Staubli VAL3: StaubliCalTool7.dtx

bool bFinish
bool bTeach1_1
bool bTeach1_2
bool bTeach1_3
bool bTeach1_4
bool bTeach2_2_1
bool bTeach2_2_2
bool bTeach2_3_1
bool bTeach2_3_2
bool bTeach2_3_3
bool bTeach3_1
bool bTeach3_2
public bool bUpLoad
configRx cConfigSame
jointRx jTest = {j1=43.06, j2=91.68, j3=-102.32, j4=-44.78, j5=56.91, j6=19.1}
mdesc mNomSpeed = {blend=cartesian}
mdesc mSlow = {vel=2, tmax=20, blend=cartesian, leave=0, reach=0}
mdesc mSpeed = {blend=cartesian, leave=0, reach=0}
num nMount = 1
num nOffsetRx
num nOffsetRy
num nOffsetRz
num nOffsetX
num nOffsetY
num nOffsetZ
num nS1[4]
num nS2[4]
num nS3[4]
num nS4[4]
num nScX
num nScY
num nScZ
pointRx p1_1 = {fatherId=world[0]}
pointRx p1_2 = {fatherId=world[0]}
pointRx p1_3 = {fatherId=world[0]}
pointRx p1_4 = {fatherId=world[0]}
pointRx p2_2_1 = {fatherId=world[0]}
pointRx p2_2_2 = {fatherId=world[0]}
pointRx p2_3_1 = {fatherId=world[0]}
pointRx p2_3_2 = {fatherId=world[0]}
pointRx p2_3_3 = {fatherId=world[0]}
pointRx p3_1 = {fatherId=world[0]}
pointRx p3_2 = {fatherId=world[0]}
pointRx pA = {x=1125.79, y=48.029029, z=-225.08575, rx=138.637496, ry=-37.318166, rz=51.328762, fatherId=world[0]}
pointRx pB = {x=1125.79, y=48.029029, z=-225.08575, rx=-41.362504, ry=-142.681834, rz=-38.671238, fatherId=world[0]}
pointRx pGoBack[11]
  [0] = {x=1244.112691, y=114.588869, z=210.083779, rx=0.001417, ry=-179.995766, rz=-83.364715, fatherId=world[0]}
  [1] = {x=1244.112692, y=114.588869, z=206.594488, rx=0.001253, ry=-179.995669, rz=-85.661401, fatherId=world[0]}
  [2] = {x=1244.112694, y=114.588869, z=203.105197, rx=0.001086, ry=-179.99558, rz=-87.958087, fatherId=world[0]}
  [3] = {x=1244.112696, y=114.588869, z=199.615906, rx=-179.999086, ry=-0.004503, rz=89.745227, fatherId=world[0]}
  [4] = {x=1244.112697, y=114.588869, z=196.126615, rx=-179.99926, ry=-0.004579, rz=87.448541, fatherId=world[0]}
  [5] = {x=1244.112699, y=114.588869, z=192.637324, rx=-179.999438, ry=-0.004648, rz=85.151855, fatherId=world[0]}
  [6] = {x=1244.1127, y=114.588869, z=189.148033, rx=-179.999618, ry=-0.00471, rz=82.855169, fatherId=world[0]}
  [7] = {x=1244.112702, y=114.588869, z=185.658742, rx=-179.9998, ry=-0.004765, rz=80.558483, fatherId=world[0]}
  [8] = {x=1244.112703, y=114.588869, z=182.169451, rx=-179.999984, ry=-0.004812, rz=78.261797, fatherId=world[0]}
  [9] = {x=1244.112705, y=114.588869, z=178.68016, rx=179.99983, ry=-0.004852, rz=75.965111, fatherId=world[0]}
  [10] = {x=1244.112706, y=114.588869, z=175.190869, rx=179.999642, ry=-0.004884, rz=73.668424, fatherId=world[0]}
pointRx pTraj = {x=1125.79, y=48.029029, z=-225.08575, rx=138.637496, ry=-37.318166, rz=42.328762, fatherId=world[0]}
string sLanguge = "Chinese"
string sMount = "floor"
string sTitle = "激光工具标定程序"
string sTool = "flange"
public tool tTool = {x=1.417, y=48.029, z=261.326, rx=-28.407, ry=-42.029, rz=-19.448, fatherId=flange[0], ioLink=valve1}
tool tTool1 = {x=1.417, y=48.029, z=261.326, rx=-28.407, ry=-42.029, rz=-19.448, fatherId=flange[0], ioLink=valve1}
tool tTool2 = {x=-11.542702, y=1.99177, z=193.654162, rx=33.798326, ry=31.269905, rz=-56.042932, fatherId=flange[0], ioLink=valve1}
tool tTool3 = {x=-12.113679, y=2.514779, z=192.872851, rx=33.798326, ry=31.269905, rz=-56.042932, fatherId=flange[0], ioLink=valve1}
